Yaskawa INFORM job: aruba_cylinder_program2.JBI

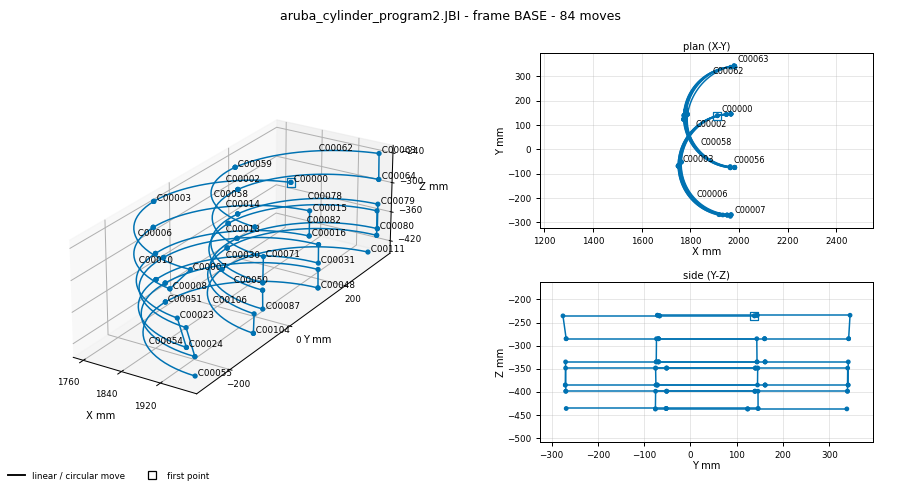
[picture p0: tool path of aruba_cylinder_program2.JBI in frame BASE, 84 of 122 moves have a stored position in this frame; points joined in program order, loops and branches not executed]
/JOB
//NAME aruba_21-05-23_cylinder_program
//POS
///NPOS 112,0,112,0,0,0
///TOOL 0
///POSTYPE BASE
///RECTAN
///RCONF 0,0,0,0,0,0,0,0,0,0,0,0,0,0,0,0,0,0,0,0,0,0,0,0
C00000=1910.805374,138.219032,-235.586000,106.047301,-90.000000,5.000000
C00001=1910.805374,138.219032,-235.586000,106.047301,-90.000000,5.000000
C00002=1804.847151,75.606057,-235.586000,140.325670,-89.999999,5.000000
C00003=1749.985059,-66.774280,-235.586000,-178.070380,-90.000000,5.000000
C00004=1749.985059,-66.774280,-235.586000,-178.070380,-90.000000,5.000000
C00005=1749.985059,-66.774280,-235.586000,-178.070380,-90.000000,5.000000
C00006=1809.269416,-210.259885,-235.586000,-136.402662,-90.000000,5.000000
C00007=1964.123044,-275.346877,-235.586000,-90.938530,-90.000000,5.000000
C00008=1917.868369,-268.447514,-284.971000,-103.399782,-89.999999,5.000000
C00009=1917.868369,-268.447514,-284.971000,-103.399782,-89.999999,5.000000
C00010=1809.935436,-211.713676,-284.971000,-136.007476,-90.000000,5.000000
C00011=1749.583414,-68.983608,-284.971000,-177.494341,-89.999999,5.000000
C00012=1749.583414,-68.983608,-284.971000,-177.494341,-89.999999,5.000000
C00013=1749.583414,-68.983608,-284.971000,-177.494341,-89.999999,5.000000
C00014=1804.888413,74.858582,-284.971000,140.474725,-90.000000,5.000000
C00015=1947.932349,143.292544,-284.971000,95.557866,-90.000000,5.000000
C00016=1947.396149,143.771403,-334.971000,95.694583,-90.000000,5.000000
C00017=1947.396149,143.771403,-334.971000,95.694583,-90.000000,5.000000
C00018=1805.924954,75.105050,-334.971000,140.243293,-90.000000,5.000000
C00019=1753.553757,-69.142352,-334.971000,-177.405543,-90.000000,5.000000
C00020=1753.553757,-69.142352,-334.971000,-177.405543,-90.000000,5.000000
C00021=1753.553757,-69.142352,-334.971000,-177.405543,-90.000000,5.000000
C00022=1811.103397,-208.756011,-334.971000,-136.356163,-90.000000,5.000000
C00023=1932.885502,-269.623207,-334.971000,-99.394426,-90.000000,5.000000
C00024=1951.055307,-270.318141,-384.971000,-94.502233,-90.000000,5.000000
C00025=1951.055307,-270.318141,-384.971000,-94.502233,-90.000000,5.000000
C00026=1821.960705,-215.828087,-384.971000,-132.973652,-89.999999,5.000000
C00027=1755.337332,-71.648560,-384.971000,-176.709276,-89.999999,5.000000
C00028=1755.337332,-71.648560,-384.971000,-176.709276,-89.999999,5.000000
C00029=1755.337332,-71.648560,-384.971000,-176.709276,-89.999999,5.000000
C00030=1805.864095,72.163968,-384.971000,140.875141,-90.000000,5.000000
C00031=1966.907277,144.834702,-384.971000,90.211125,-90.000000,5.000000
C00032=1966.424497,145.221417,-348.368460,158.362466,-71.183028,128.409256
C00033=1966.424497,145.221417,-348.368460,158.362466,-71.183028,128.409256
C00034=1815.135892,81.618659,-348.368460,170.516287,-73.092032,153.227884
C00035=1758.868193,-51.506157,-348.368460,179.529733,-73.475150,178.610026
C00036=1758.868193,-51.506157,-348.368460,179.529733,-73.475150,178.610026
C00037=1758.868193,-51.506157,-348.368460,179.529733,-73.475150,178.610026
C00038=1813.353110,-204.905937,-348.368460,-170.388574,-73.081307,-152.900122
C00039=1950.333433,-269.571661,-348.368460,-159.617006,-71.483858,-130.330207
C00040=1967.203616,-269.185645,-398.368460,-158.298210,-71.166755,-128.314971
C00041=1967.203616,-269.185645,-398.368460,-158.298210,-71.166755,-128.314971
C00042=1814.849773,-202.645210,-398.368460,-170.428104,-73.084643,-153.001442
C00043=1761.552519,-51.452927,-398.368460,179.520420,-73.475113,178.582506
C00044=1761.552519,-51.452927,-398.368460,179.520420,-73.475113,178.582506
C00045=1761.552519,-51.452927,-398.368460,179.520420,-73.475113,178.582506
C00046=1825.165223,88.648457,-398.368460,169.732631,-73.023669,151.236122
C00047=1965.878995,145.893508,-398.368460,158.406310,-71.194081,128.473819
C00048=1966.253258,146.069986,-435.651960,158.375909,-71.186421,128.429032
C00049=1966.253258,146.069986,-435.651960,158.375909,-71.186421,128.429032
C00050=1819.408689,80.794270,-435.651960,170.365739,-73.079372,152.841646
C00051=1761.998479,-52.373591,-435.651960,179.574738,-73.475317,178.743020
C00052=1761.998479,-52.373591,-435.651960,179.574738,-73.475317,178.743020
C00053=1761.998479,-52.373591,-435.651960,179.574738,-73.475317,178.743020
C00054=1827.294854,-211.521857,-435.651960,-169.450722,-72.997567,-150.531179
C00055=1966.773716,-268.374650,-435.651960,-158.332603,-71.175476,-128.365388
C00056=1963.415838,-71.360097,-234.229000,-95.383853,-90.000000,5.000000
C00057=1963.415838,-71.360097,-234.229000,-95.383853,-90.000000,5.000000
C00058=1826.683052,3.132813,-234.229000,-140.942407,-90.000000,5.000000
C00059=1788.149041,143.986421,-234.229000,175.716275,-89.999999,5.000000
C00060=1788.149041,143.986421,-234.229000,175.716275,-89.999999,5.000000
C00061=1788.149041,143.986421,-234.229000,175.716275,-89.999999,5.000000
C00062=1873.376816,294.172896,-234.229000,123.482887,-89.999999,5.000000
C00063=1979.337878,344.664409,-234.229000,90.799158,-90.000000,5.000000
C00064=1981.794114,341.634504,-284.971000,90.147398,-90.000000,5.000000
C00065=1981.794114,341.634504,-284.971000,90.147398,-90.000000,5.000000
C00066=1854.505657,289.541168,-284.971000,128.606063,-89.999999,5.000000
C00067=1783.816677,160.181911,-284.971000,171.197667,-89.999999,5.000000
C00068=1783.816677,160.181911,-284.971000,171.197667,-89.999999,5.000000
C00069=1783.816677,160.181911,-284.971000,171.197667,-89.999999,5.000000
C00070=1834.883343,-2.997765,-284.971000,-138.071367,-89.999999,5.000000
C00071=1982.109583,-73.370783,-284.971000,-90.065095,-89.999999,5.000000
C00072=1981.386588,-73.868771,-334.971000,-90.268684,-90.000000,5.000000
C00073=1981.386588,-73.868771,-334.971000,-90.268684,-90.000000,5.000000
C00074=1825.511504,4.192344,-334.971000,-141.388017,-89.999999,5.000000
C00075=1782.808202,161.229820,-334.971000,170.947768,-90.000000,5.000000
C00076=1782.808202,161.229820,-334.971000,170.947768,-90.000000,5.000000
C00077=1782.808202,161.229820,-334.971000,170.947768,-90.000000,5.000000
C00078=1852.449315,289.750467,-334.971000,129.016038,-90.000000,5.000000
C00079=1981.823638,340.854553,-334.971000,90.139940,-90.000000,5.000000
C00080=1982.305446,340.530998,-384.971000,90.009379,-90.000000,5.000000
C00081=1982.305446,340.530998,-384.971000,90.009379,-90.000000,5.000000
C00082=1850.928194,289.924830,-384.971000,129.312181,-90.000000,5.000000
C00083=1781.275226,161.272752,-384.971000,171.003719,-89.999999,5.000000
C00084=1781.275226,161.272752,-384.971000,171.003719,-89.999999,5.000000
C00085=1781.275226,161.272752,-384.971000,171.003719,-89.999999,5.000000
C00086=1825.637813,0.261147,-384.971000,-140.499099,-89.999999,5.000000
C00087=1982.037893,-74.587156,-384.971000,-90.084839,-90.000000,5.000000
C00088=1981.965863,-75.276279,-348.368460,-158.292409,-71.165281,-128.306480
C00089=1981.965863,-75.276279,-348.368460,-158.292409,-71.165281,-128.306480
C00090=1832.610423,-8.828396,-348.368460,-170.526194,-73.092857,-153.253361
C00091=1774.909146,140.405933,-348.368460,179.346084,-73.474293,178.067422
C00092=1774.909146,140.405933,-348.368460,179.346084,-73.474293,178.067422
C00093=1774.909146,140.405933,-348.368460,179.346084,-73.474293,178.067422
C00094=1840.359533,282.223263,-348.368460,169.497050,-73.001913,150.646598
C00095=1981.117594,339.615463,-348.368460,158.358795,-71.182101,128.403859
C00096=1981.953398,339.092745,-398.368460,158.292683,-71.165351,128.306880
C00097=1981.953398,339.092745,-398.368460,158.292683,-71.165351,128.306880
C00098=1831.147693,275.750162,-398.368460,170.213249,-73.066321,152.452153
C00099=1773.316170,139.287568,-398.368460,179.417157,-73.474658,178.277390
C00100=1773.316170,139.287568,-398.368460,179.417157,-73.474658,178.277390
C00101=1773.316170,139.287568,-398.368460,179.417157,-73.474658,178.277390
C00102=1830.325705,-10.068230,-398.368460,-170.567581,-73.096294,-153.359864
C00103=1964.775025,-75.245828,-398.368460,-159.671257,-71.496173,-130.416711
C00104=1963.683044,-75.685491,-436.550960,-159.754127,-71.514876,-130.549396
C00105=1963.683044,-75.685491,-436.550960,-159.754127,-71.514876,-130.549396
C00106=1831.933277,-12.541818,-436.550960,-170.379445,-73.080534,-152.876739
C00107=1771.399006,123.522149,-436.550960,-179.652728,-73.475567,-178.973508
C00108=1771.399006,123.522149,-436.550960,-179.652728,-73.475567,-178.973508
C00109=1771.399006,123.522149,-436.550960,-179.652728,-73.475567,-178.973508
C00110=1831.226640,276.569748,-436.550960,170.172244,-73.062772,152.347716
C00111=1964.923113,337.768520,-436.550960,159.635549,-71.488074,130.359742
///POSTYPE PULSE
///PULSE
EX00000=92160
EX00001=184320
EX00002=276480
EX00003=368640
///POSTYPE PULSE
///PULSE
EC00000=0
EC00001=0
EC00002=0
EC00003=0
EC00004=0
EC00005=0
EC00006=0
EC00007=0
EC00008=0
EC00009=0
EC00010=0
EC00011=0
EC00012=0
EC00013=0
EC00014=0
EC00015=0
EC00016=0
EC00017=0
EC00018=0
EC00019=0
EC00020=0
EC00021=0
EC00022=0
EC00023=0
EC00024=0
EC00025=0
EC00026=0
EC00027=0
EC00028=0
EC00029=0
EC00030=0
EC00031=0
EC00032=0
EC00033=0
EC00034=0
EC00035=0
EC00036=0
EC00037=0
EC00038=0
EC00039=0
EC00040=0
EC00041=0
EC00042=0
EC00043=0
EC00044=0
EC00045=0
EC00046=0
EC00047=0
EC00048=0
EC00049=0
EC00050=0
EC00051=0
EC00052=0
EC00053=0
EC00054=0
EC00055=0
EC00056=184320
EC00057=184320
EC00058=184320
EC00059=184320
EC00060=184320
EC00061=184320
EC00062=184320
EC00063=184320
EC00064=184320
EC00065=184320
EC00066=184320
EC00067=184320
EC00068=184320
EC00069=184320
EC00070=184320
EC00071=184320
EC00072=184320
EC00073=184320
EC00074=184320
EC00075=184320
EC00076=184320
EC00077=184320
EC00078=184320
EC00079=184320
EC00080=184320
EC00081=184320
EC00082=184320
EC00083=184320
EC00084=184320
EC00085=184320
EC00086=184320
EC00087=184320
EC00088=184320
EC00089=184320
EC00090=184320
EC00091=184320
EC00092=184320
EC00093=184320
EC00094=184320
EC00095=184320
EC00096=184320
EC00097=184320
EC00098=184320
EC00099=184320
EC00100=184320
EC00101=184320
EC00102=184320
EC00103=184320
EC00104=184320
EC00105=184320
EC00106=184320
EC00107=184320
EC00108=184320
EC00109=184320
EC00110=184320
EC00111=184320
//INST
///DATE 2023/05/23 11:20
///ATTR SC,RW,RJ
////FRAME BASE
///GROUP1 RB1,ST1
NOP
MOVJ P009 EX000 VJ=15.00
MOVJ P009 VJ=15.00
MOVJ C00000 EC00000 VJ=15.0
CALL JOB:SPYON
MOVC C00001 EC00001 V=150.0
MOVC C00002 EC00002 V=150.0
MOVC C00003 EC00003 V=150.0
MOVL C00004 EC00004 V=150.0
MOVC C00005 EC00005 V=150.0
MOVC C00006 EC00006 V=150.0
MOVC C00007 EC00007 V=150.0
MOVL C00008 EC00008 V=150.0
MOVC C00009 EC00009 V=150.0
MOVC C00010 EC00010 V=150.0
MOVC C00011 EC00011 V=150.0
MOVL C00012 EC00012 V=150.0
MOVC C00013 EC00013 V=150.0
MOVC C00014 EC00014 V=150.0
MOVC C00015 EC00015 V=150.0
MOVL C00016 EC00016 V=150.0
MOVC C00017 EC00017 V=150.0
MOVC C00018 EC00018 V=150.0
MOVC C00019 EC00019 V=150.0
MOVL C00020 EC00020 V=150.0
MOVC C00021 EC00021 V=150.0
MOVC C00022 EC00022 V=150.0
MOVC C00023 EC00023 V=150.0
MOVL C00024 EC00024 V=150.0
MOVC C00025 EC00025 V=150.0
MOVC C00026 EC00026 V=150.0
MOVC C00027 EC00027 V=150.0
MOVL C00028 EC00028 V=150.0
MOVC C00029 EC00029 V=150.0
MOVC C00030 EC00030 V=150.0
MOVC C00031 EC00031 V=150.0
MOVL C00032 EC00032 V=150.0
MOVC C00033 EC00033 V=150.0
MOVC C00034 EC00034 V=150.0
MOVC C00035 EC00035 V=150.0
MOVL C00036 EC00036 V=150.0
MOVC C00037 EC00037 V=150.0
MOVC C00038 EC00038 V=150.0
MOVC C00039 EC00039 V=150.0
MOVL C00040 EC00040 V=150.0
MOVC C00041 EC00041 V=150.0
MOVC C00042 EC00042 V=150.0
MOVC C00043 EC00043 V=150.0
MOVL C00044 EC00044 V=150.0
MOVC C00045 EC00045 V=150.0
MOVC C00046 EC00046 V=150.0
MOVC C00047 EC00047 V=150.0
MOVL C00048 EC00048 V=150.0
MOVC C00049 EC00049 V=150.0
MOVC C00050 EC00050 V=150.0
MOVC C00051 EC00051 V=150.0
MOVL C00052 EC00052 V=150.0
MOVC C00053 EC00053 V=150.0
MOVC C00054 EC00054 V=150.0
MOVC C00055 EC00055 V=150.0
CALL JOB:SPYOF
MOVJ P009 VJ=15.00
MOVL P009 EX00000 V=150.0
MOVJ P009 VJ=15.00
MOVL P009 EX00001 V=150.0
MOVJ C00056 EC00056 VJ=15.0
CALL JOB:SPYON
MOVC C00057 EC00057 V=150.0
MOVC C00058 EC00058 V=150.0
MOVC C00059 EC00059 V=150.0
MOVL C00060 EC00060 V=150.0
MOVC C00061 EC00061 V=150.0
MOVC C00062 EC00062 V=150.0
MOVC C00063 EC00063 V=150.0
MOVL C00064 EC00064 V=150.0
MOVC C00065 EC00065 V=150.0
MOVC C00066 EC00066 V=150.0
MOVC C00067 EC00067 V=150.0
MOVL C00068 EC00068 V=150.0
MOVC C00069 EC00069 V=150.0
MOVC C00070 EC00070 V=150.0
MOVC C00071 EC00071 V=150.0
MOVL C00072 EC00072 V=150.0
MOVC C00073 EC00073 V=150.0
MOVC C00074 EC00074 V=150.0
MOVC C00075 EC00075 V=150.0
MOVL C00076 EC00076 V=150.0
MOVC C00077 EC00077 V=150.0
MOVC C00078 EC00078 V=150.0
MOVC C00079 EC00079 V=150.0
MOVL C00080 EC00080 V=150.0
MOVC C00081 EC00081 V=150.0
MOVC C00082 EC00082 V=150.0
MOVC C00083 EC00083 V=150.0
MOVL C00084 EC00084 V=150.0
MOVC C00085 EC00085 V=150.0
MOVC C00086 EC00086 V=150.0
MOVC C00087 EC00087 V=150.0
MOVL C00088 EC00088 V=150.0
MOVC C00089 EC00089 V=150.0
MOVC C00090 EC00090 V=150.0
MOVC C00091 EC00091 V=150.0
MOVL C00092 EC00092 V=150.0
MOVC C00093 EC00093 V=150.0
MOVC C00094 EC00094 V=150.0
MOVC C00095 EC00095 V=150.0
MOVL C00096 EC00096 V=150.0
MOVC C00097 EC00097 V=150.0
MOVC C00098 EC00098 V=150.0
MOVC C00099 EC00099 V=150.0
MOVL C00100 EC00100 V=150.0
MOVC C00101 EC00101 V=150.0
MOVC C00102 EC00102 V=150.0
MOVC C00103 EC00103 V=150.0
MOVL C00104 EC00104 V=150.0
MOVC C00105 EC00105 V=150.0
MOVC C00106 EC00106 V=150.0
MOVC C00107 EC00107 V=150.0
MOVL C00108 EC00108 V=150.0
MOVC C00109 EC00109 V=150.0
MOVC C00110 EC00110 V=150.0
MOVC C00111 EC00111 V=150.0
CALL JOB:SPYOF
MOVJ P009 VJ=15.00
MOVL P009 EX00002 V=150.0
MOVJ P009 VJ=15.00
MOVL P009 EX00003 V=150.0
END
